FUNCTION_BLOCK RetriggerEventBasic (* Basic Function Block Type *)
  (* Standard: 61499-2 *)
  (* Version 0.0, 6/24/2026, Schneider Electric, Template *)
  PACKAGE SE.Nereda;
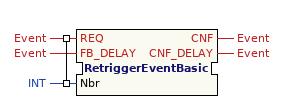
  EVENT_INPUT
    REQ WITH Nbr; (* Normal Execution Request *)
    FB_DELAY;
  END_EVENT
  EVENT_OUTPUT
    CNF; (* Execution Confirmation *)
    CNF_DELAY;
  END_EVENT
  VAR_INPUT
    Nbr : INT;
  END_VAR
  VAR
    i : INT;
  END_VAR
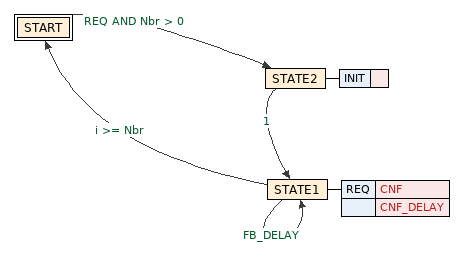
  EC_STATES
    START; (* Initial State *)
    STATE1 : REQ -> CNF, -> CNF_DELAY;
    STATE2 : INIT;
  END_STATES
  EC_TRANSITIONS
    START TO STATE2 := REQ AND Nbr > 0;
    STATE1 TO STATE1 := FB_DELAY;
    STATE1 TO START := i >= Nbr;
    STATE2 TO STATE1 := 1;
  END_TRANSITIONS
  ALGORITHM INIT IN ST: (* Initialization algorithm *)
;
i := 0;
  END_ALGORITHM
  ALGORITHM REQ IN ST: (* Normally executed algorithm *)
;
i := i + 1;
FB_DELAY := FALSE;
  END_ALGORITHM
END_FUNCTION_BLOCK
